FUNCTION_BLOCK E_CALIBRATE_SQ (* Sequential two-point calibration (offset then scale) with ECC-enforced order. *)
  (* Standard: 61499-1 *)
  (* Version 1.0, 2026-06-01, Meisterschulen am Ostbahnhof *)
  PACKAGE OSCAT::Basic::POUs::Engineering::measurements;
  (* Documentation:
  Formula
    Y = (X + OFFSET) * SCALE Calibration (Two-Point, ECC-Enforced)
    - Offset (EICO): Apply low reference, set Y_Offset to desired output, fire EICO
   OFFSET := Y_Offset / SCALE - X → after CO, Y always equals Y_Offset (independent of SCALE)
   - Scale (EICS): Apply high reference, set Y_Scale to desired output, fire EICS
   Calculates SCALE and OFFSET decoupled using both reference points → after CS, the line passes exactly through both points
    Note: Both Y_Offset and Y_Scale are target values on the output side.
    - REQ (normal operation) is always possible, even between CO and CS
   - EICS is only reachable after offset calibration (state WAIT_CS)
   - EICO can be repeated at any time to re-calibrate offset
    ECC State Machine
    START --REQ--> REQ --1--> START       (normal operation) START -EICO-> CO  --1--> WAIT_CS     (offset calibrated) WAIT_CS -REQ--> REQ --1--> WAIT_CS  (operation with offset only) WAIT_CS -EICO-> CO  --1--> WAIT_CS  (re-calibrate offset) WAIT_CS -EICS-> CS  --1--> START     (scale calibrated, done) Key Difference vs. CALIBRATE
      Feature |  CALIBRATE |  E_CALIBRATE_SQ |  
    CO formula |  OFFSET := Y_Offset - X |  OFFSET := Y_Offset / SCALE - X |  
    Y after CO |  Y = Y_Offset * SCALE
   (only correct when SCALE = 1) |  Y = Y_Offset
   (always correct) |  
    Order enforcement |  None (SimpleFB) |  ECC-enforced (CO before CS) |  
    Trigger |  BOOL inputs (CO, CS) |  Events (EICO, EICS) |  
     Example
   Scenario: 4–20 mA pressure sensor via logiBUS (0–10 V, normalized to 0.0..1.0).
   Desired output range: 0.0..500.0
      Step |  Action |  Result |  
    1 |  Apply 4 mA (X=0.0), set Y_Offset=0.0, fire EICO |  OFFSET = 0/1 − 0 = 0 |  
    2 |  Apply 20 mA (X=1.0), set Y_Scale=500.0, fire EICS |  SCALE = 500/(1+0) = 500 |  
     Output: Y = (X + 0) * 500 = X * 500 = 0..500 ✓
  *)
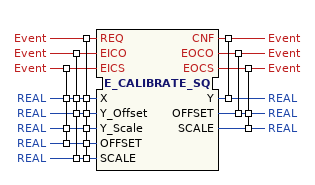
  EVENT_INPUT
    REQ WITH X, Y_Offset, Y_Scale, OFFSET, SCALE; (* Normal Execution Request (berechnet Y) *)
    EICO WITH X, Y_Offset, SCALE; (* Calibrate Offset (speichert OFFSET := Y_Offset / SCALE - X) *)
    EICS WITH X, Y_Scale, OFFSET; (* Calibrate Scale (speichert SCALE und korrigiert OFFSET basierend auf beiden Punkten) *)
  END_EVENT
  EVENT_OUTPUT
    CNF WITH Y; (* Execution Confirmed *)
    EOCO WITH OFFSET; (* Offset Calibrated *)
    EOCS WITH SCALE, OFFSET; (* Scale Calibrated *)
  END_EVENT
  VAR_INPUT
    X : REAL; (* Raw input value *)
    Y_Offset : REAL; (* Target output Y at low calibration point (offset) *)
    Y_Scale : REAL; (* Target output Y at high calibration point (scale) *)
  END_VAR
  VAR_OUTPUT
    Y : REAL; (* Calibrated output: Y = (X + OFFSET) * SCALE *)
  END_VAR
  VAR_IN_OUT
    OFFSET : REAL := 0.0; (* Stored offset value *)
    SCALE : REAL := 1.0; (* Stored scale value *)
  END_VAR
  VAR
    X_LOW_INT : REAL; (* Stored raw value at CO *)
    Y_LOW_INT : REAL; (* Stored target value at CO *)
  END_VAR
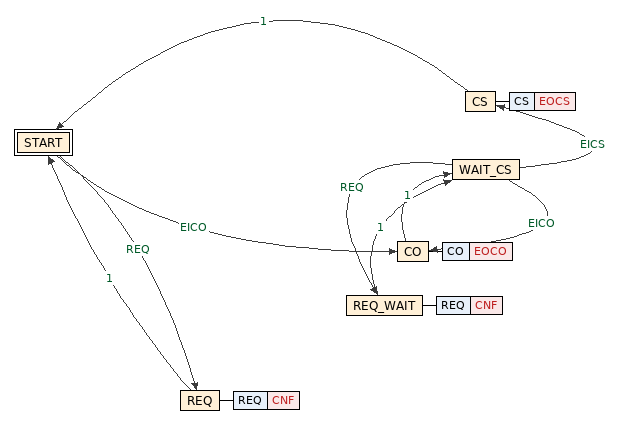
  EC_STATES
    START;
    REQ : REQ -> CNF;
    CO : CO -> EOCO;
    WAIT_CS;
    REQ_WAIT : REQ -> CNF;
    CS : CS -> EOCS;
  END_STATES
  EC_TRANSITIONS
    START TO REQ := REQ;
    REQ TO START := 1;
    START TO CO := EICO;
    CO TO WAIT_CS := 1;
    WAIT_CS TO REQ_WAIT := REQ;
    REQ_WAIT TO WAIT_CS := 1;
    WAIT_CS TO CS := EICS;
    CS TO START := 1;
    WAIT_CS TO CO := EICO;
  END_TRANSITIONS
  ALGORITHM REQ IN ST:
(* calculate calibrated output *)
Y := (X + OFFSET) * SCALE;
  END_ALGORITHM
  ALGORITHM CO IN ST:
X_LOW_INT := X;
Y_LOW_INT := Y_Offset;
IF SCALE <> 0.0 THEN
	OFFSET := Y_Offset / SCALE - X;
ELSE
	OFFSET := Y_Offset - X;
END_IF;
  END_ALGORITHM
  ALGORITHM CS IN ST:
IF (X - X_LOW_INT) <> 0.0 THEN
	SCALE := (Y_Scale - Y_LOW_INT) / (X - X_LOW_INT);
	IF SCALE <> 0.0 THEN
		OFFSET := Y_LOW_INT / SCALE - X_LOW_INT;
	END_IF;
END_IF;
  END_ALGORITHM
END_FUNCTION_BLOCK
